Staubli VAL3: clear.pgx

public program clear(screen& x_scr, num x_nX, num x_nY)
  local num i
  local num lLen
begin
  //-----------------------------------------------------------------------
  //Header begin 开头
  //Description of program  程序描述
  //  Erase the pY line from the column pX of the userPage.
  //  在用户界面中，擦除pX列中的PY行
  //Input parameters  输入参数
  //  num x_nX :
  //    role : Cursor column  作用：光标列
  //    possible value : 0 to 39  可能的值：0到39
  //  num x_nY :
  //    role : Cursor row     作用：光标行
  //    possible value : 0 to 13  可能的值：0到39
  //
  //Example 例子
  //  call clear(scrMy,15,8)
  //
  //History  历史
  //  Creation : 28-04-08 - f.Rob
  //
  //  Modified : 22 Aug 2011 - J. Cook  Added user screens
  //Header end 结束
  //-----------------------------------------------------------------------
  call typeLen(x_scr, x_nX,x_nY," ",40-x_nX)
  gotoxy(x_scr, x_nX,x_nY)
end
